TYPE E_OpClState :
(
	UNDEFINED,
	Closed,
	Open
)USINT;
END_TYPE

(* stored: Version 1.1.0.1, ProductVersion 3.1.4020.6
   DUT E_OpClState: Id {61c5e088-a74c-4c3f-aae4-f167d5cf8d0e} *)
